INTERFACE I_ActuatorWorkBase EXTENDS I_ActuatorBase

{attribute 'monitoring' := 'call'}
PROPERTY isInBasePos : BOOL
GET
END_GET
END_PROPERTY

{attribute 'monitoring' := 'call'}
PROPERTY isInWorkPos : BOOL
GET
END_GET
END_PROPERTY

METHOD public moveToBasePos : BOOL
VAR_INPUT
END_VAR
END_METHOD

METHOD public moveToWorkPos : BOOL
VAR_INPUT
END_VAR
END_METHOD

END_INTERFACE

(* stored: Version 1.1.0.1, ProductVersion 3.1.4024.3
   Itf I_ActuatorWorkBase: Id {429acf1f-cf78-427f-bf14-9e27e58ec8e6}
   Property isInBasePos: Id {8a0e9d16-dce0-43cd-bdd7-5e28c38773b4}
   Get Get: Id {f3ab26b9-6c0b-466e-8e8b-b1f0af801ae0}
   Property isInWorkPos: Id {c2dab2e5-900f-4eab-a351-cac1f6726a53}
   Get Get: Id {060c5c35-f011-4b66-9f4e-6ab14b996d88}
   Method moveToBasePos: Id {e0be16fa-848e-49c9-84b2-5359cf72f017}
   Method moveToWorkPos: Id {a426d756-d2f8-420b-aa58-a7a5b31ba1e8} *)
